FUNCTION_BLOCK StorageSkill (* Basic FB with empty ECC *)
  (* Standard: 61499-2 *)
  (* Version 1.0, 2021-09-15, dorofeev *)
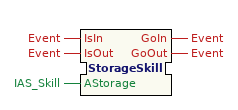
  EVENT_INPUT
    IsIn;
    IsOut;
  END_EVENT
  EVENT_OUTPUT
    GoIn;
    GoOut;
  END_EVENT
  SOCKETS
    AStorage : IAS_Skill;
  END_SOCKETS
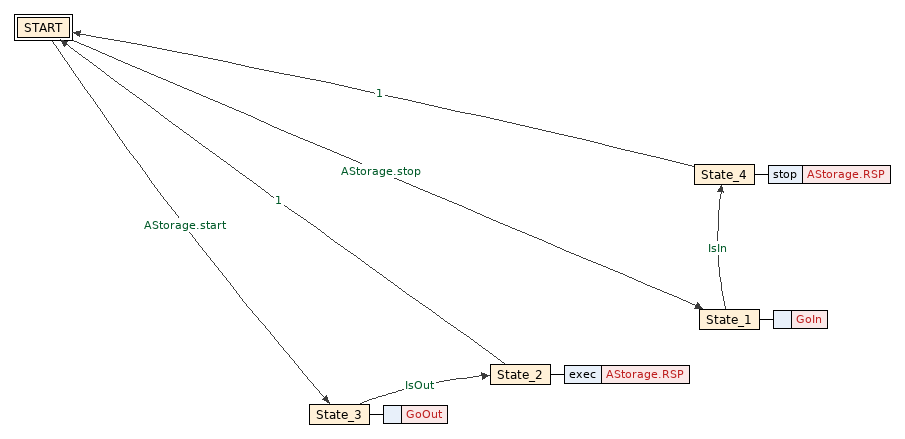
  EC_STATES
    START; (* Initial State *)
    State_1 : -> GoIn;
    State_3 : -> GoOut;
    State_2 : exec -> AStorage.RSP;
    State_4 : stop -> AStorage.RSP;
  END_STATES
  EC_TRANSITIONS
    State_1 TO State_4 := IsIn;
    State_3 TO State_2 := IsOut;
    START TO State_3 := AStorage.start;
    State_2 TO START := 1;
    START TO State_1 := AStorage.stop;
    State_4 TO START := 1;
  END_TRANSITIONS
  ALGORITHM exec IN ST: (* New Algorithm *)
AStorage.currentState := "Executing";
  END_ALGORITHM
  ALGORITHM stop IN ST: (* New Algorithm *)
AStorage.currentState := "Idle";
  END_ALGORITHM
END_FUNCTION_BLOCK
